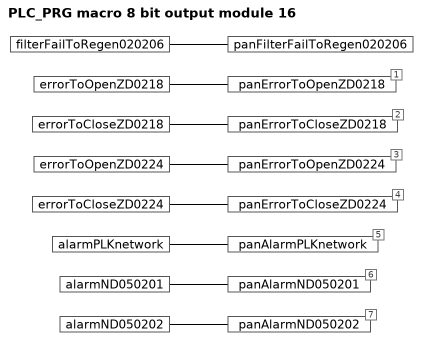
[picture p48: PLC_PRG macro 8 bit output module 16 (CFC)]
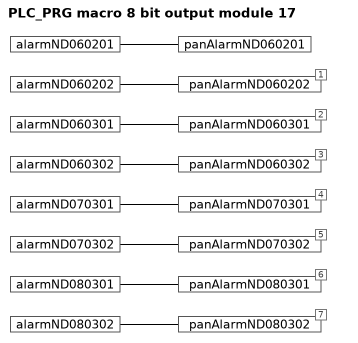
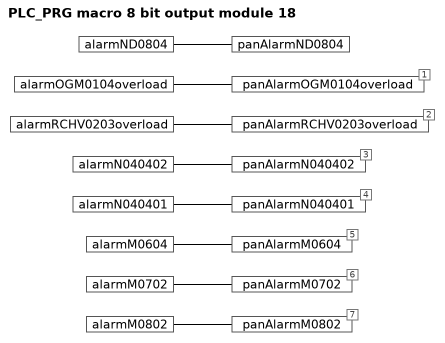
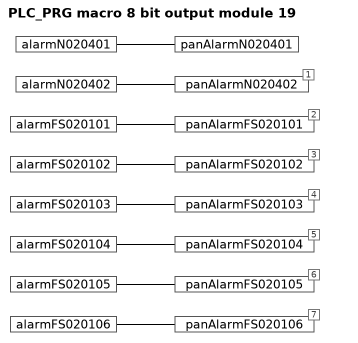
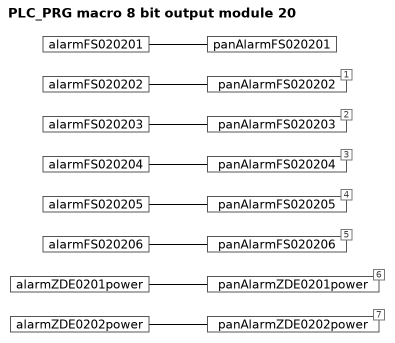
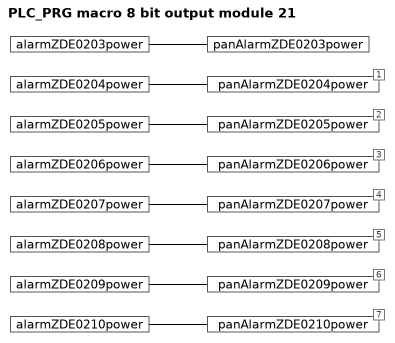
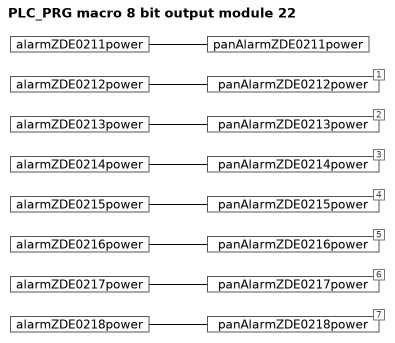
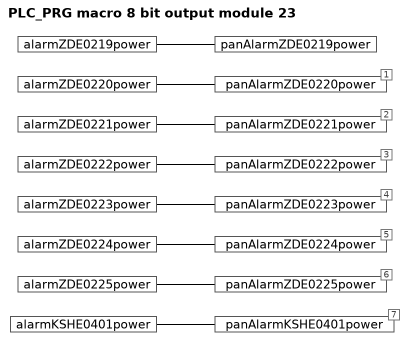
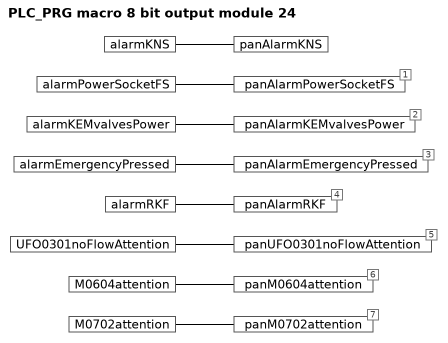
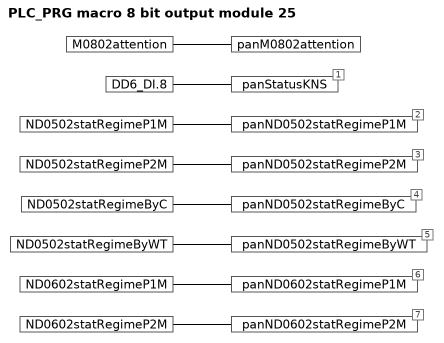
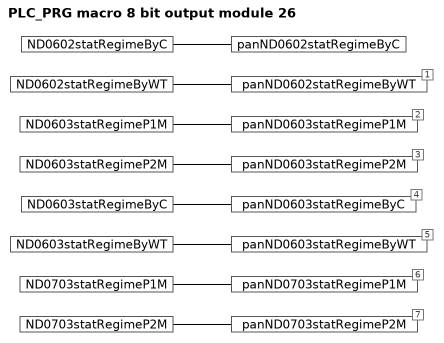
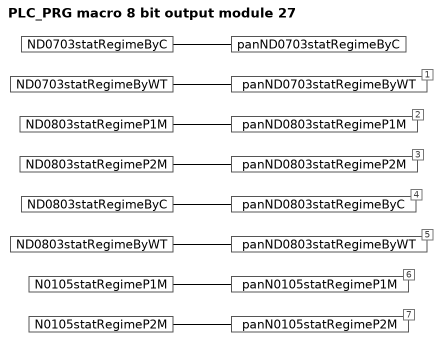
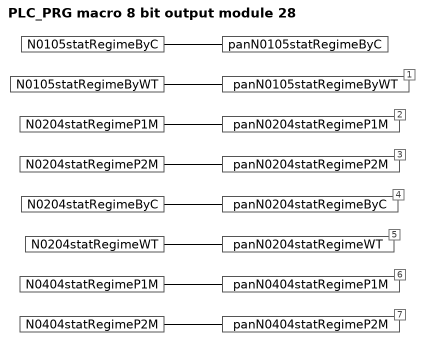
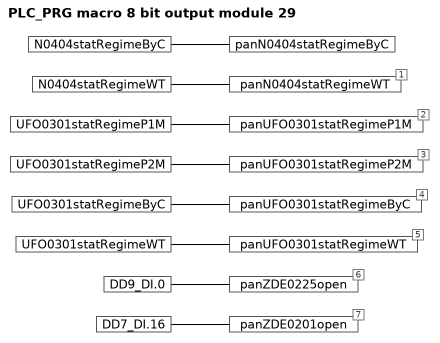
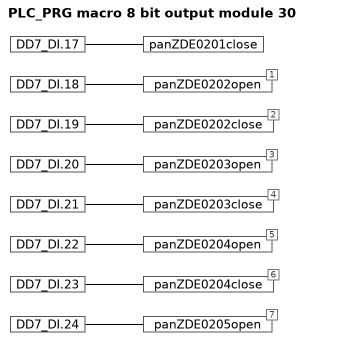
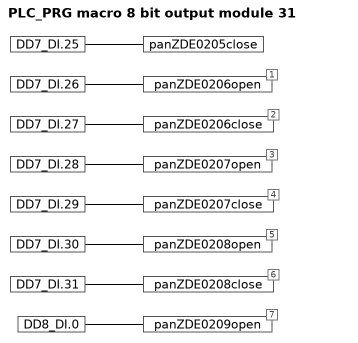
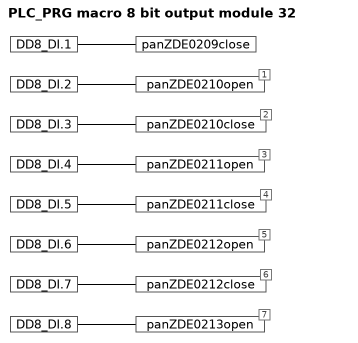
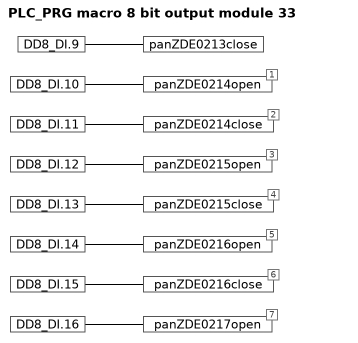
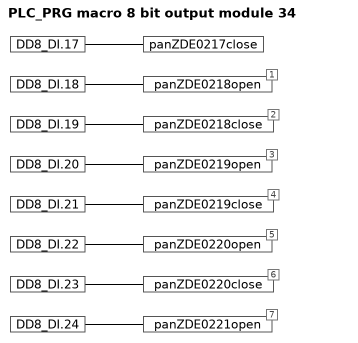
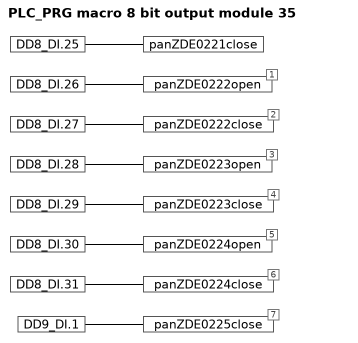
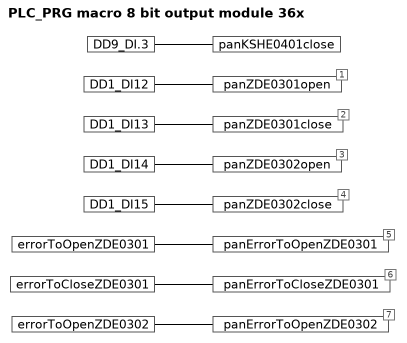
[picture p68: PLC_PRG macro 8 bit output module 36x (CFC)]
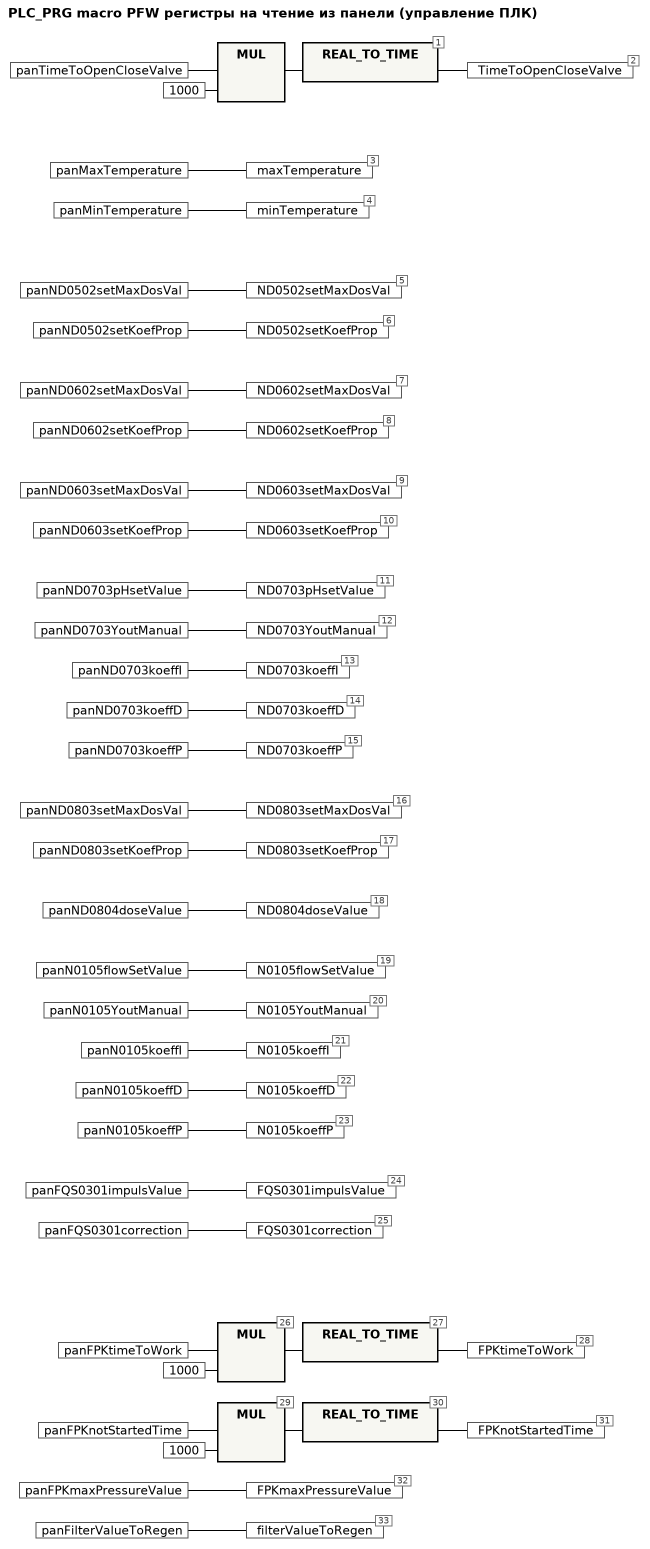
[picture p69: PLC_PRG macro PFW регистры на чтение из панели (управление ПЛК) (CFC)]
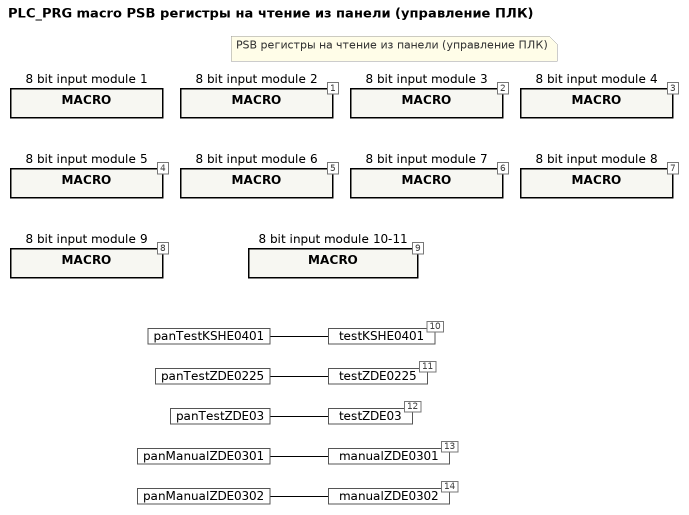
[picture p70: PLC_PRG macro PSB регистры на чтение из панели (управление ПЛК) (CFC)]
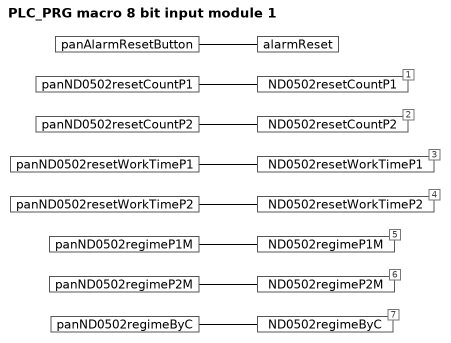
[picture p71: PLC_PRG macro 8 bit input module 1 (CFC)]
